// TIA Portal V20 export
TYPE "LKinCtrl_typePnPLinCmdSeqParameter"
   STRUCT
      start : "LKinCtrl_typePnPLinPointParameter";   // Parameter for start position
      postStart : "LKinCtrl_typePnPLinPointParameter";   // Parameter for post start motion
      intermediate : "LKinCtrl_typePnPLinPointParameter";   // Parameter for intermediate motion
      preTarget : "LKinCtrl_typePnPLinPointParameter";   // Parameter for pre target motion
      target : "LKinCtrl_typePnPLinPointParameter";   // Parameter for target motion
      numberOfUsedCmd : DInt;   // Number of used commands
   END_STRUCT;
   // start.transitionParameter[1] := -1.0;
   // postStart.transitionParameter[1] := -1.0;
   // intermediate.transitionParameter[1] := -1.0;
   // preTarget.transitionParameter[1] := -1.0;
   // target.transitionParameter[1] := -1.0;
END_TYPE
